FUNCTION TryConvert_LWORD_TO_LREAL : BOOL
VAR_INPUT
	in : LWORD;
	out : REFERENCE TO LREAL;
END_VAR

out := LWORD_TO_LREAL(in);
TryConvert_LWORD_TO_LREAL := TRUE;

END_FUNCTION

(* stored: Version 1.1.0.1, ProductVersion 3.1.4024.12
   POU TryConvert_LWORD_TO_LREAL: Id {d0d8b997-4053-47a4-bd5b-eb4184000aba}, SpecialFunc None *)
